// TIA Portal V20 export
// export: Created 2025-12-01T14:56:22.2234201Z, ExportSetting None, DisplayName Totally Integrated Automation Portal, DisplayVersion V20 Update 3, DisplayName TIA Portal Openness, DisplayVersion V20 Update 3, DisplayName TIA Portal Version Control Interface, DisplayVersion V20 Update 3, DisplayName STEP 7 Professional, DisplayVersion V20 Update 3, DisplayName STEP 7 Safety, DisplayVersion V20 Update 2, DisplayName WinCC Basic/Comfort/Advanced, DisplayVersion V20 Update 3, DisplayName WinCC Professional, DisplayVersion V20 Update 3, DisplayName WinCC Unified, DisplayVersion V20 Update 3
TYPE "NDD_Ordenes"
   STRUCT
      Operacion_EntradaPaleta : Bool;
      Operacion_PaletizarPaleta : Bool;
      Operacion_EvacuarPaleta : Bool;
      Operacion_TElev_Garras : Bool;
      Operacion_TElev_Horquilla : Bool;
      Operacion_Horq_Garra : Bool;
      Operacion_Garra_Elev : Bool;
      Libre_07 : Bool;
      TElev_PaletaVacia : Bool;
      TElev_PaletaCargada : Bool;
      TElev_Enfradar : Bool;
      TElev_Paletizar : Bool;
      Libre_13 : Bool;
      Libre_14 : Bool;
      Libre_15 : Bool;
      TElev_SinUT : Bool;
      TElev_CodigoEnfardado : Int;
      TElev_CotaAltura : Int;
   END_STRUCT;
END_TYPE
